// TIA Portal project "Soru1" (V15)

(* hardware
DEVICE "S7-1200 station_1"  S7-1200 Station
   slot 0: "Rack_0"  S7-1200 Rack  Rack  V1.0
   slot 1: "PLC_1"  CPU 1214C DC/DC/Rly  6ES7 214-1HG40-0XB0  V4.2
*)

// ===== PLC "PLC_1"  CPU 1214C DC/DC/Rly =====

VAR_GLOBAL   // PLC tag table "Default tag table"
   "1.btn" AT %I0.0 : Bool;
   "1. motor" AT %Q0.0 : Bool;
   "Stop" AT %I0.1 : Bool;
   "2.motor" AT %Q0.1 : Bool;
END_VAR

ORGANIZATION_BLOCK "Main"   // OB1, LAD, ProgramCycle
TITLE = "Main Program Sweep (Cycle)"
{ S7_Optimized_Access := 'TRUE' }
VERSION : 0.1
   VAR_INPUT
      Initial_Call : Bool;   // Initial call of this OB
      Remanence : Bool;   // =True, if remanent data are available
   END_VAR
BEGIN

REGION Network 1
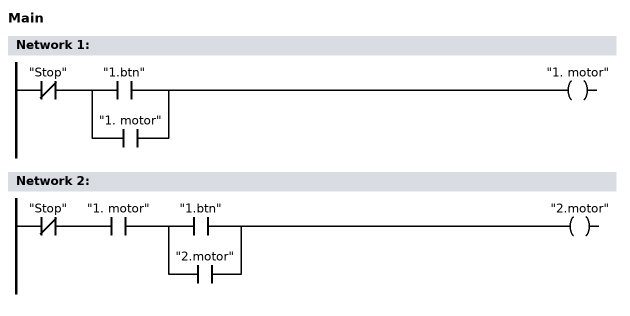
   RUNG wire#powerrail
      I_Contact( "Stop" )
      wire#w1
      Contact( "1.btn" )
      wire#w2
      Coil( "1. motor" )
   END_RUNG
   RUNG wire#w1
      Contact( "1. motor" )
   END_RUNG wire#w2
   // the same network as SCL:
   "1. motor" := NOT "Stop" AND ("1.btn" OR "1. motor");
END_REGION

REGION Network 2
   RUNG wire#powerrail
      I_Contact( "Stop" )
      Contact( "1. motor" )
      wire#w1
      Contact( "1.btn" )
      wire#w2
      Coil( "2.motor" )
   END_RUNG
   RUNG wire#w1
      Contact( "2.motor" )
   END_RUNG wire#w2
   // the same network as SCL:
   "2.motor" := NOT "Stop" AND "1. motor" AND ("1.btn" OR "2.motor");
END_REGION
END_ORGANIZATION_BLOCK